// Utils functions deprecated — topping logic moved into EventTracker
// Kept as placeholder to avoid broken references
PROGRAM UTILS_DEPRECATED
VAR
    placeholder : BOOL := FALSE;
END_VAR

// placeholder
placeholder := placeholder;

END_PROGRAM

(* stored: Version 1.1.0.1, ProductVersion 3.1.4024.15
   POU Utils_DEPRECATED: Id {a1c7b6d1-0000-4f2a-a111-1234567890ab} *)
